Fanuc KAREL source: kd00023.KL

-- PROVISIONAL review KL for V1013-1; original PC SHA256 80d5262321aaf1f92628f48fe503d1d81fcbc868716ca28af9dec3d0383c4861
-- Incomplete behavior may be omitted. Consult companion uncertainty JSON. Do not deploy.
PROGRAM KD00023
%NOLOCKGROUP
VAR
  I : INTEGER
  J : INTEGER
  B : BOOLEAN
  R : REAL
  S : STRING[80]
  SAVED : INTEGER
BEGIN
  -- UNRESOLVED_PC offsets 5-17; opcodes 21,23
  -- UNRESOLVED_PC offsets 22-26; opcodes 7F
END KD00023
